// ---- FB/41_PosCom/FB/FB_013_POS_Comparition.TcPOU
FUNCTION_BLOCK FB_013_POS_Comparition
VAR_IN_OUT
	arstCamCtrl          : ARRAY[*] OF  ST_EL5131_CamCtrl; //1-X轴 2-Y轴
	fbstIJP                :  ST_IJP;
	stAxis               :ARRAY[*] OF  ST_AXIS;
END_VAR
//VAR_INPUT
//	nXAxisId:UDINT;
//	nYAxisId:UDINT;
//	nZAxisId:UDINT;
//END_VAR
VAR
  	bAxisInPosStart: ARRAY [1..3] OF BOOL;
	bAxisInPosEnd:  ARRAY [1..3] OF BOOL;
    tonWriteR:ARRAY [1..5] OF TON;
    stepWriteR:ARRAY [1..4] OF INT;
  	bInStartZone: BOOL;
	bInEndZone:BOOL;
	i:INT;
	bEx_TrigEl5131Rtrig:r_trig;
	bEx_TrigStartRtrig:r_trig;
    bEx_TrigEndRtrig:r_trig;
	bEx_TrigEl5131Ftrig:f_trig;
    nAxisIdStep:int;
END_VAR


{region "位置比较"}
bEx_TrigEl5131Rtrig(CLK:=fbstIJP.bEx_TrigEl5131 , Q=> );
IF bEx_TrigEl5131Rtrig.Q THEN
        tonWriteR[1](IN:= FALSE);
		tonWriteR[2](IN:= FALSE);
		tonWriteR[3](IN:= FALSE);
		tonWriteR[5](IN := FALSE);
END_IF	 
		   
IF fbstIJP.bEx_TrigEl5131 THEN
  FOR i:=1 TO fbstIJP.EL5131_CamCtrlMax BY 1 DO
	// 起点比较触发   
	bEx_TrigStartRtrig(CLK:=bInStartZone , Q=> );
	// 起点触发后延时
	tonWriteR[5](IN := (fbstIJP.bEx_Trigfb AND fbstIJP.bEx_TrigHfb) , PT := fbstIJP.tEndPosDelay );
	// 延时后终点比较触发
	bEx_TrigEndRtrig(CLK:=bInEndZone AND tonWriteR[5].Q, Q=> );
	// 起点位置比较
	IF arstCamCtrl[i].udiAxisId1<>0 THEN	 
	   bAxisInPosStart[1] := ABS(stAxis[arstCamCtrl[i].udiAxisId1].State.rActPos - arstCamCtrl[i].rPosStart1) < fbstIJP.rPosTolerance ;
	ELSE
	   bAxisInPosStart[1]:=TRUE;
	END_IF
	IF arstCamCtrl[i].udiAxisId2<>0 THEN
       bAxisInPosStart[2] := ABS(stAxis[arstCamCtrl[i].udiAxisId2].State.rActPos - arstCamCtrl[i].rPosStart2) < fbstIJP.rPosTolerance ;
	ELSE
	   bAxisInPosStart[2]:=TRUE;
	END_IF
    IF arstCamCtrl[i].udiAxisId3<>0 THEN
       bAxisInPosStart[3] := ABS(stAxis[arstCamCtrl[i].udiAxisId3].State.rActPos - arstCamCtrl[i].rPosStart2) < fbstIJP.rPosTolerance;
	ELSE
	   bAxisInPosStart[3]:=TRUE;
    END_IF 
	// 终点位置比较
	IF arstCamCtrl[i].udiAxisId1<>0 THEN
       bAxisInPosEnd[1] := ABS(stAxis[1].State.rActPos - arstCamCtrl[i].rPosEnd1) < fbstIJP.rPosTolerance;
	ELSE
	   bAxisInPosStart[1]:=TRUE;
	END_IF
	IF arstCamCtrl[i].udiAxisId2<>0 THEN
       bAxisInPosEnd[2] := ABS(stAxis[2].State.rActPos - arstCamCtrl[i].rPosEnd2) < fbstIJP.rPosTolerance;
	ELSE
	   bAxisInPosStart[2]:=TRUE;
	END_IF
	IF arstCamCtrl[i].udiAxisId3<>0 THEN
       bAxisInPosEnd[3] := (ABS(stAxis[3].State.rActPos - arstCamCtrl[i].rPosEnd2) < fbstIJP.rPosTolerance) ;
    ELSE
	   bAxisInPosStart[3]:=TRUE;
    END_IF 	
    bInStartZone := bAxisInPosStart[1] AND bAxisInPosStart[2] AND bAxisInPosEnd[3];
	bInEndZone   := bEx_TrigEndRtrig.Q AND bAxisInPosEnd[1] AND bAxisInPosEnd[2] AND bAxisInPosEnd[3];	 
    // 起点开
    IF bEx_TrigStartRtrig.Q AND arstCamCtrl[1].bCamCtrlStartEn THEN
       fbstIJP.bEl5131_Trig := TRUE;
       fbstIJP.bEl5131_TrigH := TRUE;
	   arstCamCtrl[1].bCamCtrlStartEn:=FALSE;
	END_IF
	// 终点关
    IF  bEx_TrigEndRtrig.Q AND arstCamCtrl[1].bCamCtrlEndEn THEN
           fbstIJP.bEl5131_Trig := FALSE;
           fbstIJP.bEl5131_TrigH := FALSE;
        END_IF		
  END_FOR
ELSE
    // —— 复位 —— 
    tonWriteR[5](IN := FALSE);		 
    fbstIJP.bEl5131_Trig := FALSE;
    fbstIJP.bEl5131_TrigH := FALSE;
END_IF
{endregion}

END_FUNCTION_BLOCK

// ---- POUs/15_Gear/ProgGear.TcPOU
PROGRAM ProgGear
VAR
	fbGear:ARRAY[1..2] OF FB_Gear;
	i:UINT;
	GearTrig:R_TRIG;
	PlatY_TO_RollR1Rtrig:R_TRIG;
	RollY1_TO_RollYRtrig:R_TRIG;
	RollZ1_TO_RollZ2Rtrig:R_TRIG;
	RollR1_TO_RollR2Rtrig:R_TRIG;
	PlatY_TO_RollR1Ftrig:F_TRIG;
	RollY1_TO_RollYFtrig:F_TRIG;
	RollZ1_TO_RollZ2Ftrig:F_TRIG;
	RollR1_TO_RollR2Ftrig:F_TRIG;
	mcGearInDyn			:MC_GearInDyn;	
	mcGearOut			:MC_GearOut;
	bTest				:BOOL;
	bTestOut			:BOOL;
	rRatio				:LREAL:=1.0;
	mcMoveVel			:MC_MoveVelocity;
	bExe				:BOOL;
	blink				:BLINK;
END_VAR

A_01_R1_TO_R2();
A_01_R1_TO_R3();

ACTION A_01_R1_TO_R2:
// 轴基础参数设定
arstGear[1].wstrName:=" 喷头R1轴与R2轴耦合" ;
arstGear[1].rSyncVelocity:=arstAxis[7].Pos.Par.rVel;
arstGear[1].rSyncACC:=arstAxis[7].Pos.Par.rAcc;
arstGear[1].rRatioNumerator:=1;
arstGear[1].uiRatioDenominator:=1;
arstGear[1].bStop_A:=arstAxis[7].Control.bStop_A;
// 功能块
fbGear[1](AxisRefSlave:=arAxis[8] ,AxisRefMaster:=arAxis[7],stSystem:=stSystem,stGear:=arstGear[1] , inChannelid:=1 );
END_ACTION

ACTION A_01_R1_TO_R3:
// 轴基础参数设定
arstGear[2].wstrName:=" 喷头R1轴与R3轴耦合" ;
arstGear[2].rSyncVelocity:=arstAxis[7].Pos.Par.rVel;
arstGear[2].rSyncACC:=arstAxis[7].Pos.Par.rAcc;
arstGear[2].rRatioNumerator:=1;
arstGear[2].uiRatioDenominator:=1;
arstGear[2].bStop_A:=arstAxis[7].Control.bStop_A;
// 功能块
fbGear[2](AxisRefSlave:=arAxis[9] ,AxisRefMaster:=arAxis[7],stSystem:=stSystem,stGear:=arstGear[2] , inChannelid:=2 );
END_ACTION

END_PROGRAM

// ---- FB/71_Gear/FB/FB_Gear.TcPOU
FUNCTION_BLOCK FB_Gear
VAR_IN_OUT
	stGear:ST_Gear;
	AxisRefMaster:AXIS_REF;
	AxisRefSlave:AXIS_REF;
	stSystem:ST_System;
//	arrfbSetAlarm: ARRAY[1..3] OF FB_SetError;
END_VAR
VAR_INPUT
	inChannelid:INT;
END_VAR
VAR
	fbGearIn:MC_GearIn;
	fbGearInDyn:MC_GearInDyn;
	fbGearout:MC_GearOut;
	fbGearoutTrig:R_TRIG;
	arrfbSetAlarm: ARRAY[1..3] OF FB_SetError;
	i:UINT;
	statr: BOOL;
END_VAR

fbGearInDyn(
	Master:= AxisRefMaster, 
	Slave:= AxisRefSlave, 
	Enable:= stGear.bGearIn(*arstGear[2].bGearIn*), 
	GearRatio:=stGear.rRatioNumerator, 
	Acceleration:= , 
	Deceleration:= , 
	Jerk:= , 
	BufferMode:= , 
	Options:= , 
	InGear=> , 
	Busy=> , 
	Active=> , 
	CommandAborted=> , 
	Error=> stGear.bError, 
	ErrorID=> );
//fbGearIn(
//	Master:= stGear.AxisRefMaster, 
//	Slave:= stGear.AxisRefSlave, 
//	Execute:= stGear.bGearIn, 
//	RatioNumerator:= stGear.rRatioNumerator, 
//	RatioDenominator:= stGear.uiRatioDenominator, 
//	Acceleration:= , 
//	Deceleration:=, 
//	Jerk:= , 
//	BufferMode:= , 
//	Options:= , 
//	InGear=> , 
//	Busy=> , 
//	Active=> , 
//	CommandAborted=> , 
//	Error=> stGear.bError, 
//	ErrorID=> );
stGear.bInSyncing:=AxisRefSlave.Status.Coupled;
fbGearout(
	Slave:=  AxisRefSlave(*stGear.AxisRefSlave*) , 
	Execute:= stGear.bGearOut , 
	Options:= , 
	Done=> stGear.bnoInSyncing, 
	Busy=> , 
	Error=> stGear.bError, 
	ErrorID=> );
//fbGearoutTrig(CLK:=fbGearout.Done , Q=> );
//	IF fbGearoutTrig.Q THEN
//		stGear.bGearin:=FALSE;
//	END_IF
IF fbGearIn.Error THEN
	stGear.bError:=TRUE;
	stGear.arErrorID[1]:=TRUE;
//ELSIF fbGearInPos.Error THEN
	//stGear.arErrorID[2]:=TRUE;
ELSIF fbGearout.Error THEN
	stGear.bError:=TRUE;
	stGear.arErrorID[2]:=TRUE;
END_IF
// 耦合报错
arrfbSetAlarm[1](
	bEnable:= TRUE, 
	iErrorID:= 80+3*(inChannelid-1), 
	bExecute:= stGear.arErrorID[1], 
	bReset:= stSystem.bReset, 
	strErrorInfoEN:= 'Gear_in Alm', 
	wstrErrorInfoCN:="耦合错误" , 
	enumErrorClass:= 6, 
    );
// 耦合报错
arrfbSetAlarm[3](
	bEnable:= TRUE, 
	iErrorID:= 80+3*(inChannelid-1)+2, 
	bExecute:= stGear.arErrorID[3], 
	bReset:= stSystem.bReset, 
	strErrorInfoEN:= 'Gear_in Alm', 
	wstrErrorInfoCN:=" 解耦错误" , 
	enumErrorClass:= 6, 
    );
IF stSystem.bReset THEN
	stGear.bError:=FALSE;
	FOR i:=1 TO 2 BY 1 DO 
	   stGear.arErrorID[i]:=FALSE;
    END_FOR
END_IF

END_FUNCTION_BLOCK

// ---- POUs/05_气缸控制/YV_Ctrl.TcPOU
PROGRAM YV_Ctrl
VAR
	fbPOU1: ARRAY[1..4] OF FB_V_3B5;
	i:UINT;
	j:INT;
	bFirstRun: BOOL;
END_VAR

IF bFirstRun=FALSE THEN
	FOR i:=1 TO 4 BY 1 DO
		arstYV[i].bYVBw_A:=FALSE;
	END_FOR
arstYV[1].bYVFw_A:=TRUE;
arstYV[2].bYVFw_A:=TRUE;
arstYV[3].bYVFw_A:=TRUE;
arstYV[4].bYVFw_A:=TRUE;
//    bFirstRun:=TRUE;
END_IF	

ACT_01_BlowYV();   // 对中气缸

ACTION ACT_01_BlowYV:

//放料气缸(左)
IF bFirstRun=FALSE THEN
arstYV[1].bYVFw_A:=TRUE;
arstYV[1].bYVBw_A:=FALSE;
bFirstRun:=TRUE;
END_IF
// 	气缸IO关联
arstYV[1].bYVBw_In:=X000007;     //  缩回
arstYV[1].bYVFw_In:=X000006 ;    //  伸出
//stYV[3].bYVBw_Out:=Y00105;   
//stYV[3].bYVFw_Out:=Y00106;   
Y000005:=arstYV[1].bYVBw_Out (*AND NOT X00102) OR NOT X00102 *) ;       // 缩回
Y000004:=arstYV[1].bYVFw_Out (*OR (X00102 AND arstYV[1].bYVBw_Out)*) ;   // 伸出
// 功能块
fbPOU1[1](fbstYV:=arstYV[1],stSystem:=stSystem,inChannelid:=1);
END_ACTION

END_PROGRAM

// ---- FB/05_YV/FB_V_3B5.TcPOU
FUNCTION_BLOCK FB_V_3B5
VAR_IN_OUT
	fbstYV:ST_YV;
	stSystem:ST_System;
END_VAR
VAR_INPUT
	inChannelid:INT;
END_VAR

VAR
	tonYVFwCHK:ton;
	tonYVFwTimeOut:ton;
	tonYVBwCHK:ton;
	tonYV1BwTimeOut:ton;
	arError :ARRAY  [1..4]OF BOOL;
	i: UINT;
	arrfbSetAlarm: ARRAY[1..3] OF FB_SetError;
END_VAR


(********************************************YV1*****************************************)
//气缸伸出
fbstYV.bYVFw_Out :=fbstYV.bYVFw_A  ;
tonYVFwCHK(IN:=fbstYV.bYVFw_Out AND fbstYV.bYVFw_In  , 
PT:=TIME#5MS ,
 Q=>fbstYV.bYVFw_OK , 
ET=> );
//伸出超时报警
tonYVFwTimeOut(IN:=fbstYV.bYVFw_Out AND NOT  fbstYV.bYVFw_OK , 
PT:=TIME#3S , 
Q=>arError[1] , 
ET=> );


//气缸缩回
fbstYV.bYVBw_Out :=fbstYV.bYVBw_A ;
tonYVBwCHK(IN:=fbstYV.bYVBw_Out AND fbstYV.bYVBw_In ,
 PT:=TIME#5MS ,
 Q=>fbstYV.bYVBw_OK , 
ET=> );
//缩回超时报警
tonYV1BwTimeOut(IN:=fbstYV.bYVBw_out AND NOT fbstYV.bYVBw_OK ,
 PT:=TIME#3S , 
 Q=>arError[2] , 
ET=> );

IF arError[1]=TRUE THEN
	fbstYV.bError:=TRUE;
	fbstYV.udiError:=1;
	fbstYV.arErrorID[0]:=TRUE;	
ELSIF arError[2]=TRUE THEN
	fbstYV.bError:=TRUE;
	fbstYV.udiError:=2;
	fbstYV.arErrorID[1]:=TRUE;		
//同时检测到伸出缩回到位信号
ELSIF fbstYV.bYVFw_In AND fbstYV.bYVBw_In THEN
	fbstYV.bError:=TRUE;
	fbstYV.udiError:=3;
	fbstYV.arErrorID[2]:=TRUE;	
ELSE
	fbstYV.bError:=FALSE;
    fbstYV.udiError:=0;
	FOR i:=1 TO 4 BY 1 DO 
	  fbstYV.arErrorID[i]:=0;		 
	END_FOR
END_IF
// 伸出报错
arrfbSetAlarm[1](
	bEnable:= TRUE, 
	iErrorID:= 90+3*(inChannelid-1), 
	bExecute:= fbstYV.arErrorID[1], 
	bReset:= stSystem.bReset, 
	strErrorInfoEN:= 'Bw_out Alm', 
	wstrErrorInfoCN:="伸出超时报警" , 
	enumErrorClass:= 6, 
    );
// 伸出报错
arrfbSetAlarm[1](
	bEnable:= TRUE, 
	iErrorID:= 90+3*(inChannelid-1), 
	bExecute:= fbstYV.arErrorID[1], 
	bReset:= stSystem.bReset, 
	strErrorInfoEN:= 'Fw_out Alm', 
	wstrErrorInfoCN:="缩回超时报警" , 
	enumErrorClass:= 6, 
    );
// 伸出报错
arrfbSetAlarm[1](
	bEnable:= TRUE, 
	iErrorID:= 90+3*(inChannelid-1), 
	bExecute:= fbstYV.arErrorID[1], 
	bReset:= stSystem.bReset, 
	strErrorInfoEN:= 'Fw_BW Alm', 
	wstrErrorInfoCN:="限位同时触发报警", 
	enumErrorClass:= 6, 
    );

END_FUNCTION_BLOCK

// ---- POUs/14_Bump/Pump.TcPOU
PROGRAM Pump
VAR
  iPumpStep   : INT := 0;  // 状态机步骤
  rRelPos     : REAL;    // 定量容积距离  mm
  rRelVel     : REAL;    // 流速线速度  mm/s
  posEdgePump : R_TRIG;  // 仅保留 M21(启动) 的上升沿触发器，M26(停止) 改为直接电平判断
	rTrigPrintStop: INT;
	Q: INT;
	ton01:ton;
END_VAR

// ==========================================
// 1. 触发信号边缘检测
// ==========================================
posEdgePump(CLK := stPump.bEx_PumpTrigOn); // M21 启动信号检测

// ==========================================
// 1.5 异常中断拦截 (防漏液与防抽气保护)
// ==========================================
IF stIJP.bStopExe THEN
    // 核心逻辑：只在“准备挤出”或“正在挤出”的阶段（步号 9 到 20 之间）才干预
    IF iPumpStep >= 9 AND iPumpStep <= 20 THEN
        
//        // 1. 立即撤销所有可能的运动触发信号
      arstaxis[10].Pos.Ctrl.bGo_A := FALSE;   // 撤销定量运动
      arstaxis[10].Control.bJogCw_A := FALSE; // 撤销匀速运动
        
//        // 2. 向底层轴发送停止指令
       arstaxis[10].Control.bStop_A := TRUE;
        
//        // 3. 强制状态机跳转到过渡状态25
//        // (状态25会等待电机停稳，然后自动进入29执行回抽)
        iPumpStep := 25;
        
//    // 如果 iPumpStep = 0 (静止状态) 
//    // 或者 iPumpStep >= 25 (已经处于停机缓冲或回抽状态)
//    // 则什么都不做，完美避免了闲置时抽空气的问题
   END_IF
END_IF

// ==========================================
// 2. 注射泵控制状态机
// ==========================================
CASE iPumpStep OF
    0:  // --- 等待状态 (Idle) ---
        // M21上升沿触发，进入流程1
        IF posEdgePump.Q THEN
            iPumpStep := 5;
        END_IF
    
    5:  // --- 流程1准备：刷新参数并计算 ---
        stPump.bEx_PumpTrigOn := FALSE; 					// 【防呆】阅后即焚：复位M21启动信号，防止HMI按钮卡死  
        stPump.rJogVol_A := stPump.rVol_Process1;
        stPump.rJogVel_A := stPump.rVel_Process1;
        ACT_Calc();              					// 调用Action，立刻计算出 rRelPos 和 rRelVel
        iPumpStep := 6;
	
    6: // --- 流程1：快速注入 (发送指令) ---
        arstaxis[10].Pos.Par.rVel   := rRelVel;
        arstaxis[10].Pos.Par.rPos    := rRelPos;
        arstaxis[10].Pos.Par.bRelEnable := TRUE;         	
		iPumpStep := 10;
        
    10: // --- 流程1：快速注入 (发送指令) ---   
        arstaxis[10].Pos.Ctrl.bGo_A   := TRUE;  	// 触发运动      
        // 等待底层确认收到指令并脱离静止状态
        //IF arAXIS[10].Status.Moving OR NOT arAXIS[10].Status.StandStill THEN
            iPumpStep := 11; 
        //END_IF
    11: // --- 流程1：快速注入 (等待完成) ---
        // 确保到位后再进行下一步
       // IF (NOT arAXIS[10].Status.Moving) AND (arAXIS[10].Status.StandStill) AND arAXIS[10].Status.InTargetPosition THEN
	   IF arstaxis[10].Pos.State.bGo_OK THEN
            arstaxis[10].Pos.Ctrl.bGo_A := FALSE; 	// 复位执行信号
            iPumpStep := 19;                        // 无缝进入流程2准备阶段
        END_IF
        
    19: // --- 流程2准备：刷新参数并计算 ---
        stPump.rJogVel_A := stPump.rVel_Process2;      
        ACT_Calc();              					// 立刻计算出新的连续运动速度 rRelVel
        iPumpStep := 20;      
        
    20: // --- 流程2：匀速注入 (连续运动) ---
	    arstaxis[10].Control.iJogMode:=0;
        arstaxis[10].Parameter.rJogVel_A   := rRelVel;
        //arstaxis[10].Parameter.uiMoveMode := 0;
        arstaxis[10].Control.bJogCw_A     := TRUE;  // 触发连续匀速运动

        // 等待 M26 信号停止流程2
        // 【优化】直接判断电平并复位，取消上升沿依赖，防止误触漏信号
        IF stPump.bEx_PumpTrigOff THEN
            arstaxis[10].Control.bJogCw_A := FALSE;   // 取消匀速指令
            arstaxis[10].Control.bStop_A  := TRUE;    // 发送轴停止指令
            iPumpStep := 25;                        	// 进入过渡缓冲状态
        END_IF

    25: // --- 过渡状态：等待电机停稳 (安全保护) ---
        IF arstaxis[10].State.bStandStill AND NOT arstaxis[10].State.bMoving AND NOT arAXIS[10].Status.HasJob THEN
            arstaxis[10].Control.bStop_A := FALSE;    // 复位停止信号
			stPump.bEx_PumpTrigOff      := FALSE;   // 【防呆】阅后即焚：复位M26停止信号
            iPumpStep := 26;                        // 电机停稳，进入流程3准备
        END_IF
    26:
       IF ton01.Q  THEN
			iPumpStep := 27;
		END_IF    
    27: // --- 流程3准备：刷新参数并计算 ---
        stPump.rJogVol_A := stPump.rVol_Process3;
        stPump.rJogVel_A := stPump.rVel_Process3;
        
        ACT_Calc();              // 立刻计算出抽取参数
        iPumpStep := 29;      
    29:    
        arstaxis[10].Pos.Par.rVel   := rRelVel;			// 【关键】速度必须为正
        arstaxis[10].Pos.Par.rPos    := -rRelPos;		// 【关键】位移取负，实现反转抽取
        arstaxis[10].Pos.Par.bRelEnable := TRUE;  
       iPumpStep := 30; 
    30: // --- 流程3：快速抽取 (定量) ---

        arstaxis[10].Pos.Ctrl.bGo_A   := TRUE;  		// 触发运动
         
        //IF arAXIS[10].Status.Moving OR NOT arAXIS[10].Status.StandStill THEN
            iPumpStep := 31;
        //END_IF
    31: 
        IF ton01.Q  THEN
			iPumpStep := 32;
		END_IF
    32: // --- 流程3：快速抽取 (等待完成) ---
       // IF (NOT arAXIS[10].Status.Moving) AND (arAXIS[10].Status.StandStill) (*AND arAXIS[10].Status.InTargetPosition*) THEN
		IF	arstaxis[10].Pos.State.bGo_OK THEN
            arstaxis[10].Pos.Ctrl.bGo_A   := FALSE;     // 复位执行信号
            iPumpStep := 0;                             // 整个流程结束，回到待机状态
        END_IF
                         
END_CASE;
ton01(IN:=(iPumpStep=31) OR (iPumpStep=26) , PT:=T#50MS , Q=> , ET=> ); 
// ==========================================
// 3. 状态反馈给上位机 (放在最底部)
// ==========================================
stPump.iCurrentStep := iPumpStep;

ACTION ACT_Calc:
// ==========================================
// Action: ACT_Calc (容积转运动距离与速度)
// ==========================================
IF stPump.strml='2.5ml' THEN
    rRelPos := stPump.rJogVol_A / ((stPump.rInjectDia[1]/2)*(stPump.rInjectDia[1]/2)*3.1415926);
    rRelVel := stPump.rJogVel_A / 60 / ((stPump.rInjectDia[1]/2)*(stPump.rInjectDia[1]/2)*3.1415926);
ELSIF stPump.strml='5ml' THEN
    rRelPos := stPump.rJogVol_A / ((stPump.rInjectDia[2]/2)*(stPump.rInjectDia[2]/2)*3.1415926);
    rRelVel := stPump.rJogVel_A / 60 / ((stPump.rInjectDia[2]/2)*(stPump.rInjectDia[2]/2)*3.1415926);
//ELSIF stPump.strml='10ml' THEN
//    rRelPos := stPump.rJogVol_A / ((stPump.rInjectDia[3]/2)*(stPump.rInjectDia[3]/2)*3.1415926);
//    rRelVel := stPump.rJogVel_A / 60 / ((stPump.rInjectDia[3]/2)*(stPump.rInjectDia[3]/2)*3.1415926);
//ELSIF stPump.strml='30ml' THEN
//    rRelPos := stPump.rJogVol_A / ((stPump.rInjectDia[4]/2)*(stPump.rInjectDia[4]/2)*3.1415926);
//    rRelVel := stPump.rJogVel_A / 60 / ((stPump.rInjectDia[4]/2)*(stPump.rInjectDia[4]/2)*3.1415926);
END_IF
END_ACTION

END_PROGRAM

// ---- FB/61_Alarm/FB/FB_Alarm.TcPOU
FUNCTION_BLOCK FB_Alarm
VAR_OUTPUT
	//当前有报警发生
	bErrorOccur						:				BOOL					;
	//当前发生报警的最大报警等级
	enumErrorClassMax				:				Enum_ErrorClass			;(*当前的最大报警等级*)
END_VAR
VAR
	// 报警整合输出变量，不启用
	bNoStopAlarm					:               BOOL					;
   	// 不启用
	bStopAlarm						:               BOOL					;
END_VAR
VAR_OUTPUT
	//报警整合后输出动作，根据需求设定
	bAlarmAction1					:				BOOL					;
	bAlarmAction2					:				BOOL					;
	bAlarmAction3					:				BOOL					;
	bAlarmAction4					:				BOOL					;
END_VAR
VAR
	strVersion: STRING;
	i								:               INT						;
	m								:               INT						;
	n								:               INT						;
	rtrigErrorOccur					:          		R_TRIG					;
	tonErrorOccur					: 				TON						;
	ftrigClearHistory				: 				F_TRIG					;
	ftrigErrorOccur					: 				F_TRIG					;
	fbGetLocalSystemTime				:				FB_LocalSystemTime		;
	fbGetLocalAmsNetID: FB_GetLocalAmsNetId;
	binitdone: BOOL;
	Ton01: TON;
END_VAR

ACTION A_ClearHistoryError:
//手动清除历史报警数组
ftrigClearHistory(CLK:=bClearHistoryError  );
IF ftrigClearHistory.Q THEN
       FOR n:=1 TO 200 DO
             arrstHistoryError[n].iErrorID:=0;
             arrstHistoryError[n].wstrErrorMessage:="";
             arrstHistoryError[n].dtErrorTime:=DT#2024-05-11-00:00;
        END_FOR
        iHistoryErrorNum:=0;
END_IF
END_ACTION

ACTION A_Init:
//获取系统netid
fbGetLocalAmsNetID(
	bExecute:= TRUE, 
	tTimeOut:= , 
	bBusy=> , 
	bError=> , 
	nErrId=> , 
	AddrString=> , 
	AddrBytes=> );
Ton01(IN:=TRUE,PT:=TIME#50MS);
IF ton01.Q AND NOT fbGetLocalAmsNetID.bBusy THEN	
	binitdone := TRUE ;
END_IF;
END_ACTION

ACTION A_UpdateActError:
//有报警发生时，将报警数据抓取存储到当前报警数组中
rtrigErrorOccur(CLK:=bErrorOccur);
IF bErrorOccur THEN
	IF rtrigErrorOccur.Q THEN
   	 	tonErrorOccur(In:=FALSE);
	END_IF
    tonErrorOccur(In:= NOT tonErrorOccur.Q,PT:=T#1S );
    IF tonErrorOccur.Q OR rtrigErrorOccur.Q THEN
		n:=1;
        m:=1;
        FOR n:=1 TO iErrorIDMax DO
			IF arrstError[n].bErrorOccur THEN
				arrstActError[m].iErrorID := arrstError[n].iErrorID;
				arrstActError[m].wstrErrorMessage := arrstError[n].wstrErrorMessage;						
				arrstActError[m].dtErrorTime := arrstError[n].dtErrorOccorTime;
                m:=m+1;
				IF m>30 THEN
					n:=32766;  (*exit FOR*)
				END_IF
			END_IF
         END_FOR
         IF m<30 THEN
			FOR n:=m TO 30 DO
				arrstActError[n].iErrorID:=0;
                arrstActError[n].wstrErrorMessage:="";
                arrstActError[n].dtErrorTime:=DT#2024-05-11-00:00;
             END_FOR
          END_IF
    END_IF
	//当前存在的报警数量
	iActErrorNum := m-1;
END_IF

//报警消除后，清除当前报警数组
ftrigErrorOccur(CLK:=bErrorOccur );
IF ftrigErrorOccur.Q THEN
	FOR n:=1 TO 30 DO 
		arrstActError[n].iErrorID:=0;
		arrstActError[n].wstrErrorMessage:="";
		arrstActError[n].dtErrorTime:=DT#2024-05-11-00:00;
	END_FOR
	iActErrorNum:=0;
END_IF
END_ACTION

END_FUNCTION_BLOCK
